// TwinCAT 3 PLC project TcoPneumaticsTests
// Title: TcoPneumaticsTests
// Company: Vortex.Library
// ProjectVersion: 0.6.0.913
// ProgramVersion: 3.1.4024.12
// libraries:
//   Tc2_Standard, * (Beckhoff Automation GmbH)
//   Tc2_System, * (Beckhoff Automation GmbH)
//   Tc3_Module, * (Beckhoff Automation GmbH)
//   TcoCore, 0.6.0.913 (Vortex.Library)
//   TcoPneumatics, 0.6.0.913 (Vortex.Library)
// project tree:
//   ComponentExampleImplementation/ExampleCyclinderUsage/ ExampleCylinderContext.TcPOU
//   ComponentExampleImplementation/ExampleCylinder/ ExampleCylinder.TcPOU, ExampleCylinderConfig.TcDUT, ExampleCylinderMoveTask.TcPOU, ExampleCylinderStatus.TcDUT
//   ComponentExampleImplementation/ EXAMPLE_MAIN.TcPOU
//   GVLs/ IO.TcGVL
//   / PlcTask.TcTTO
//   POUs/CylinderBaseTests/ CylinderBaseImplemented.TcPOU, DoubleCylinderBaseImplemented.TcPOU, CylinderBaseTestContext.TcPOU, DoubleCylinderBaseTestContext.TcPOU, eCyclinderBaseTests.TcDUT
//   POUs/CylinderTests/ DoubleCylinderTestContext.TcPOU, eCyclinderTests.TcDUT, CylinderTestContext.TcPOU
//   POUs/ DefaultContext.TcPOU, MAIN.TcPOU
// (motion and I/O tree: see PLC project tcopneumatics)
// real-time tasks:
//   TASK PlcTask: cycle T#10ms, priority 20, ADS port 350
//   TASK PlcTask1: cycle T#10ms, priority 21, ADS port 351

CONFIGURATION TcoPneumaticsTests
    RESOURCE PLC ON TwinCAT3
        TASK PlcTask(INTERVAL := T#10ms, PRIORITY := 20);
        PROGRAM MAIN WITH PlcTask : MAIN;
        PROGRAM EXAMPLE_MAIN WITH PlcTask : EXAMPLE_MAIN;
    END_RESOURCE
END_CONFIGURATION

// ---- ComponentExampleImplementation/ExampleCylinder/ExampleCylinderConfig.TcDUT
TYPE ExampleCylinderConfig :
STRUCT
    TimeToReachHomePosition : TIME := T#10S;
    TimeToReachWorkPosition : TIME := T#10S;
END_STRUCT
END_TYPE

// ---- ComponentExampleImplementation/ExampleCylinder/ExampleCylinderStatus.TcDUT
TYPE ExampleCylinderStatus :
STRUCT
    ActionDescription : STRING(100);
END_STRUCT
END_TYPE

// ---- POUs/CylinderBaseTests/eCyclinderBaseTests.TcDUT
{attribute 'qualified_only'}
{attribute 'strict'}
TYPE eCyclinderBaseTests :
(
    Invalid := 50,
    GetAtHome := 100,
    GetAtWork := 200
);
END_TYPE

// ---- POUs/CylinderTests/eCyclinderTests.TcDUT
{attribute 'qualified_only'}
{attribute 'strict'}
TYPE eCyclinderTests :
(
    Invalid := 25,
    StopMovement := 50,
    MoveHomeMoving := 100,
    MoveHomeMovingReached := 200,
    MoveWorkMoving := 300,
    MoveWorkMovingReached := 400,
    AbortMoveTask := 500,
    DisableHome := 600,
    DisableWork := 700,
    SuspendHome := 610,
    SuspendWork := 710,
    SuspendHomeInverted := 620,
    SuspendWorkInverted := 720,
    SuspendHomeExpression := 630,
    SuspendWorkExpression := 730
);
END_TYPE

// ---- GVLs/IO.TcGVL
{attribute 'qualified_only'}
VAR_GLOBAL
    {attribute addProperty Name "A1"}
    A1 AT %I* : ARRAY[0..7] OF BOOL;
    {attribute addProperty Name "A2"}
    A2 AT %Q* : ARRAY[0..7] OF BOOL;
END_VAR

// ---- POUs/MAIN.TcPOU
PROGRAM MAIN
VAR
    _defaultContext : DefaultContext;
    _cylinderBaseTests : CylinderBaseTestContext;
    _doubleCylinderBaseTests : DoubleCylinderBaseTestContext;
    _cylinderTests : CylinderTestContext;
    _doubleCylinderTests : DoubleCylinderTestContext;
END_VAR

_defaultContext.Run();
_cylinderTests.ProbeRun();
_doubleCylinderTests.ProbeRun();
_cylinderBaseTests.ProbeRun();
_doublecylinderBaseTests.ProbeRun();

END_PROGRAM

// ---- POUs/DefaultContext.TcPOU
FUNCTION_BLOCK DefaultContext EXTENDS TcoCore.TcoContext
VAR
    {attribute addProperty _moveHomeDefaultName "<#MOVE HOME#>"}
    {attribute addProperty _moveWorkDefaultName "<#MOVE TO WORK#>"}
    {attribute addProperty _stopDefaultName "<#STOP a#>"}
    _wpfCyclinder : TcoPneumatics.TcoCylinder(THIS^);
    {attribute addProperty _moveHomeDefaultName "<#MOVE HOME#>"}
    {attribute addProperty _moveWorkDefaultName "<#MOVE TO WORK#>"}
    {attribute addProperty _stopDefaultName "<#STOPDOUBLE#>"}
    _wpfDoubleCyclinder : TcoPneumatics.TcoDoubleCylinder(THIS^);
    {attribute addProperty NameMoveHomeTask "<#In task#>"}
    _wpfCyclinder_1 : TcoPneumatics.TcoCylinder(THIS^);
    {attribute addProperty NameMoveHomeTask "<#In task#>"}
    _wpfCyclinder_2 : TcoPneumatics.TcoCylinder(THIS^);
    {attribute addProperty NameMoveHomeTask "<#In task#>"}
    _wpfCyclinder_3 : TcoPneumatics.TcoCylinder(THIS^);
    disableSignalWork : BOOL;
    disableSignalHome : BOOL;
    suspendSignalWork : BOOL;
    suspendSignalHome : BOOL;
    refilCondition : BOOL;
END_VAR

METHOD PROTECTED Main
VAR
    ;
END_VAR
THIS^.RtcSynchronize(TRUE, '', 60);
_wpfCyclinder.Service();

_wpfCyclinder(inoAtHomePos := IO.A1[0],
    inoAtWorkPos := IO.A1[1],
    inoToHomePos := IO.A2[0],
    inoToWorkPos := IO.A2[1]);

_wpfCyclinder.AbortMoveHome(disableSignalHome);
_wpfCyclinder.AbortMoveWork(disableSignalWork);
_wpfCyclinder.SuspendMoveHome(suspendSignalHome);
_wpfCyclinder.SuspendMoveWork(suspendSignalWork);
//optional blocking options
//_wpfCyclinder.SuspendMoveWorkInverted(suspendSignalWork);	// is basicaly option how to reproduce exaxt symbol and Not condition
//_wpfCyclinder.SuspendMoveWorkExpression(NOT suspendSignalWork,'Your own msg');	// is basicaly option how to reproduce exaxt symbol and Not condition
_wpfCyclinder.Refill(T#200MS);
_wpfDoubleCyclinder.Service();

_wpfDoubleCyclinder(inoAtHomePos1 := IO.A1[0],
    inoAtHomePos2 := IO.A1[1],
    inoAtWorkPos1 := IO.A1[2],
    inoAtWorkPos2 := IO.A1[3],
    inoToHomePos := IO.A2[3],
    inoToWorkPos := IO.A2[4]);

_wpfDoubleCyclinder.AbortMoveHome(disableSignalHome);
_wpfDoubleCyclinder.AbortMoveWork(disableSignalWork);
_wpfDoubleCyclinder.SuspendMoveHome(suspendSignalHome);
_wpfDoubleCyclinder.SuspendMoveWork(suspendSignalWork);
//optional blocking options
//_wpfDoubleCyclinder.SuspendMoveWorkInverted(suspendSignalWork);	// is basicaly option how to reproduce exaxt symbol and Not condition
//_wpfDoubleCyclinder.SuspendMoveWorkExpression(NOT suspendSignalWork,'Your own msg');	// is basicaly option how to reproduce exaxt symbol and Not condition
_wpfDoubleCyclinder.Refill(T#200MS);
END_METHOD

END_FUNCTION_BLOCK

// ---- POUs/CylinderBaseTests/CylinderBaseTestContext.TcPOU
FUNCTION_BLOCK CylinderBaseTestContext EXTENDS TcoCore._internals_TcoContext
VAR
    _sut : CylinderBaseImplemented(THIS^);
    _sutInvalid : CylinderBaseImplemented(THIS^);
    _atHomeSignal : BOOL;
    _atWorkSignal : BOOL;
    _toHomeSignal : BOOL;
    _toWorkSignal : BOOL;
END_VAR
VAR
    _get_AtHome : BOOL;
    _get_AtWork : BOOL;
END_VAR

METHOD PROTECTED Main
_sut(inoAtHomePos := _atHomeSignal,
    inoAtWorkPos := _atWorkSignal,
    inoToHomePos := _toHomeSignal,
    inoToWorkPos := _toWorkSignal);

CASE _testId OF
    eCyclinderBaseTests.Invalid:
        _sutInvalid.AtHome;
        _sutInvalid.AtWork;
        _sutInvalid.Restore();
        _sutInvalid.Stop();
    eCyclinderBaseTests.GetAtHome:
        _get_AtHome := _sut.AtHome;
    eCyclinderBaseTests.GetAtWork:
        _get_AtWork := _sut.AtWork;
END_CASE
END_METHOD

END_FUNCTION_BLOCK

// ---- POUs/CylinderBaseTests/CylinderBaseImplemented.TcPOU
FUNCTION_BLOCK CylinderBaseImplemented EXTENDS TcoPneumatics.TcoCylinder

SUPER^(inoAtHomePos := inoAtHomePos,
    inoAtWorkPos := inoAtWorkPos,
    inoToHomePos := inoToHomePos,
    inoToWorkPos := inoToWorkPos);

PROPERTY MoveHomeTask : TcoCore.ITcoTask
GET
END_GET
SET
END_SET
END_PROPERTY

PROPERTY MoveWorkTask : TcoCore.ITcoTask
GET
END_GET
SET
END_SET
END_PROPERTY

PROPERTY StopTask : TcoCore.ITcoTask
GET
END_GET
SET
END_SET
END_PROPERTY

END_FUNCTION_BLOCK

// ---- POUs/CylinderBaseTests/DoubleCylinderBaseTestContext.TcPOU
FUNCTION_BLOCK DoubleCylinderBaseTestContext EXTENDS TcoCore._internals_TcoContext
VAR
    _sut : DoubleCylinderBaseImplemented(THIS^);
    _sutInvalid : DoubleCylinderBaseImplemented(THIS^);
    _atHomeSignal : BOOL;
    _atWorkSignal : BOOL;
    _toHomeSignal : BOOL;
    _toWorkSignal : BOOL;
END_VAR
VAR
    _get_AtHome : BOOL;
    _get_AtWork : BOOL;
END_VAR

METHOD PROTECTED Main
_sut(inoAtHomePos1 := _atHomeSignal,
    inoAtHomePos2 := _atHomeSignal,
    inoAtWorkPos1 := _atWorkSignal,
    inoAtWorkPos2 := _atWorkSignal,
    inoToHomePos := _toHomeSignal,
    inoToWorkPos := _toWorkSignal);

CASE _testId OF
    eCyclinderBaseTests.Invalid:
        _sutInvalid.AtHome;
        _sutInvalid.AtWork;
        _sutInvalid.Restore();
        _sutInvalid.Stop();
    eCyclinderBaseTests.GetAtHome:
        _get_AtHome := _sut.AtHome;
    eCyclinderBaseTests.GetAtWork:
        _get_AtWork := _sut.AtWork;
END_CASE
END_METHOD

END_FUNCTION_BLOCK

// ---- POUs/CylinderBaseTests/DoubleCylinderBaseImplemented.TcPOU
FUNCTION_BLOCK DoubleCylinderBaseImplemented EXTENDS TcoPneumatics.TcoDoubleCylinderBase

SUPER^(inoAtHomePos1 := inoAtHomePos1,
    inoAtHomePos2 := inoAtHomePos2,
    inoAtWorkPos1 := inoAtWorkPos1,
    inoAtWorkPos2 := inoAtWorkPos2,
    inoToHomePos := inoToHomePos,
    inoToWorkPos := inoToWorkPos);

PROPERTY MoveHomeTask : TcoCore.ITcoTask
GET
END_GET
SET
END_SET
END_PROPERTY

PROPERTY MoveWorkTask : TcoCore.ITcoTask
GET
END_GET
SET
END_SET
END_PROPERTY

PROPERTY StopTask : TcoCore.ITcoTask
GET
END_GET
SET
END_SET
END_PROPERTY

END_FUNCTION_BLOCK

// ---- POUs/CylinderTests/CylinderTestContext.TcPOU
FUNCTION_BLOCK CylinderTestContext EXTENDS TcoCore._internals_TcoContext
VAR
    {attribute addProperty _moveHomeDefaultName "<#MOVE HOME SWEET HOME#>"}
    {attribute addProperty _moveWorkDefaultName "<#MOVE TO WORK HARD WORK#>"}
    {attribute addProperty _stopDefaultName "<#STOP AND THINK#>"}
    _sut : TcoPneumatics.TcoCylinder(THIS^);
    _sutInvalid : TcoPneumatics.TcoCylinder(THIS^);
    _atHomeSignal : BOOL;
    _moveHomeSignal : BOOL;
    _atWorkSignal : BOOL;
    _moveWorkSignal : BOOL;
END_VAR
VAR
    _moveHomeDone : BOOL;
    _moveWorkDone : BOOL;
    _disableSignal : BOOL;
    _suspendSignal : BOOL;
    _expresionMessage : STRING;
END_VAR

METHOD PROTECTED Main
_sut(inoAtHomePos := _atHomeSignal,
    inoAtWorkPos := _atWorkSignal,
    inoToHomePos := _moveHomeSignal,
    inoToWorkPos := _moveWorkSignal);

CASE _testId OF
    eCyclinderTests.Invalid:
        _sutInvalid.Stop();
        _sutInvalid.MoveToHome();
        _sutInvalid.MoveToWork();
        _sutInvalid.Service();
        _sutInvalid.AtHome;
        _sutInvalid.AtWork;
        _sutInvalid.AbortMoveHome(_disableSignal);
        _sutInvalid.AbortMoveHome(_disableSignal);
        _sutInvalid.Config.TimeToReachHomePosition := T#1MS;
        _sutInvalid.Config.TimeToReachWorkPosition := T#1MS;
        _sutInvalid.Status.ActionDescription;
    eCyclinderTests.StopMovement:
        _sut.Stop();
    eCyclinderTests.MoveHomeMoving:
        _moveHomeDone := _sut.MoveToHome().Done;
    eCyclinderTests.MoveHomeMovingReached:
        _moveHomeDone := _sut.MoveToHome().Done;
    eCyclinderTests.MoveWorkMoving:
        _moveWorkDone := _sut.MoveToWork().Done;
    eCyclinderTests.MoveWorkMovingReached:
        _moveWorkDone := _sut.MoveToWork().Done;
    eCyclinderTests.AbortMoveTask:
        _sut.MoveHomeTask.Abort();
    eCyclinderTests.DisableHome:
        _sut.AbortMoveHome(_disableSignal);
    eCyclinderTests.DisableWork:
        _sut.AbortMoveWork(_disableSignal);
    eCyclinderTests.SuspendHome:
        _sut.SuspendMoveHome(_suspendSignal);
    eCyclinderTests.SuspendWork:
        _sut.SuspendMoveWork(_suspendSignal);
    eCyclinderTests.SuspendHomeInverted:
        _sut.SuspendMoveHomeInverted(_suspendSignal);
    eCyclinderTests.SuspendWorkInverted:
        _sut.SuspendMoveWorkInverted(_suspendSignal);
    eCyclinderTests.SuspendHomeExpression:
        _sut.SuspendMoveHomeExpression(_suspendSignal, _expresionMessage);
    eCyclinderTests.SuspendWorkExpression:
        _sut.SuspendMoveWorkExpression(_suspendSignal, _expresionMessage);
END_CASE
END_METHOD

END_FUNCTION_BLOCK

// ---- POUs/CylinderTests/DoubleCylinderTestContext.TcPOU
FUNCTION_BLOCK DoubleCylinderTestContext EXTENDS TcoCore._internals_TcoContext
VAR
    {attribute addProperty _moveHomeDefaultName "<#MOVE HOME SWEET HOME#>"}
    {attribute addProperty _moveWorkDefaultName "<#MOVE TO WORK HARD WORK#>"}
    {attribute addProperty _stopDefaultName "<#STOP AND THINK#>"}
    _sut : TcoPneumatics.TcoDoubleCylinder(THIS^);
    _sutInvalid : TcoPneumatics.TcoDoubleCylinder(THIS^);
    _atHomeSignal : BOOL;
    _moveHomeSignal : BOOL;
    _atWorkSignal : BOOL;
    _moveWorkSignal : BOOL;
END_VAR
VAR
    _moveHomeDone : BOOL;
    _moveWorkDone : BOOL;
    _disableSignal : BOOL;
    _suspendSignal : BOOL;
    _expresionMessage : STRING;
END_VAR

METHOD PROTECTED Main
_sut(inoAtHomePos1 := _atHomeSignal,
    inoAtHomePos2 := _atHomeSignal,
    inoAtWorkPos1 := _atWorkSignal,
    inoAtWorkPos2 := _atWorkSignal,
    inoToHomePos := _moveHomeSignal,
    inoToWorkPos := _moveWorkSignal);

CASE _testId OF
    eCyclinderTests.Invalid:
        _sutInvalid.Stop();
        _sutInvalid.MoveToHome();
        _sutInvalid.MoveToWork();
        _sutInvalid.Service();
        _sutInvalid.AtHome;
        _sutInvalid.AtWork;
        _sutInvalid.AbortMoveHome(_disableSignal);
        _sutInvalid.AbortMoveHome(_disableSignal);
        _sutInvalid.Config.TimeToReachHomePosition := T#1MS;
        _sutInvalid.Config.TimeToReachWorkPosition := T#1MS;
        _sutInvalid.Status.ActionDescription;
    eCyclinderTests.StopMovement:
        _sut.Stop();
    eCyclinderTests.MoveHomeMoving:
        _moveHomeDone := _sut.MoveToHome().Done;
    eCyclinderTests.MoveHomeMovingReached:
        _moveHomeDone := _sut.MoveToHome().Done;
    eCyclinderTests.MoveWorkMoving:
        _moveWorkDone := _sut.MoveToWork().Done;
    eCyclinderTests.MoveWorkMovingReached:
        _moveWorkDone := _sut.MoveToWork().Done;
    eCyclinderTests.AbortMoveTask:
        _sut.MoveHomeTask.Abort();
    eCyclinderTests.DisableHome:
        _sut.AbortMoveHome(_disableSignal);
    eCyclinderTests.DisableWork:
        _sut.AbortMoveWork(_disableSignal);
    eCyclinderTests.SuspendHome:
        _sut.SuspendMoveHome(_suspendSignal);
    eCyclinderTests.SuspendWork:
        _sut.SuspendMoveWork(_suspendSignal);
    eCyclinderTests.SuspendHomeInverted:
        _sut.SuspendMoveHomeInverted(_suspendSignal);
    eCyclinderTests.SuspendWorkInverted:
        _sut.SuspendMoveWorkInverted(_suspendSignal);
    eCyclinderTests.SuspendHomeExpression:
        _sut.SuspendMoveHomeExpression(_suspendSignal, _expresionMessage);
    eCyclinderTests.SuspendWorkExpression:
        _sut.SuspendMoveWorkExpression(_suspendSignal, _expresionMessage);
END_CASE
END_METHOD

END_FUNCTION_BLOCK

// ---- ComponentExampleImplementation/EXAMPLE_MAIN.TcPOU
PROGRAM EXAMPLE_MAIN
VAR
    _context : ExampleCylinderContext;
END_VAR

_context.Run();

END_PROGRAM

// ---- ComponentExampleImplementation/ExampleCyclinderUsage/ExampleCylinderContext.TcPOU
FUNCTION_BLOCK ExampleCylinderContext EXTENDS TcoCore.TcoContext
VAR
    _exampleCylinder : ExampleCylinder(THIS^);
    _atHome : BOOL;
    _atWork : BOOL;
    _toHome : BOOL;
    _toWork : BOOL;
END_VAR

(*~
    <docu>
        <summary>
            Main method of the TcoContext. This is the entry point of any control logic that belongs to this context.
            The call of this method is ensured by calling the <c>InstanceName.Run()</c> method, and it must not be called explicitly.
            This method is abstract, and it must be overridden in derived block.
        </summary>
    </docu>
~*)
METHOD PROTECTED Main
VAR_INST
    _state : INT;
END_VAR
_exampleCylinder(inoAtHomePos := _atHome,
    inoAtWorkPos := _atWork,
    inoToHomePos := _toHome,
    inoToWorkPos := _toWork);

CASE _state OF
    0:
        IF (_exampleCylinder.MoveToHome().Done) THEN
            _state := 10;
        END_IF
    10:
        IF (_exampleCylinder.MoveToWork().Done) THEN
            _state := 0;
        END_IF
END_CASE
END_METHOD

END_FUNCTION_BLOCK

// ---- ComponentExampleImplementation/ExampleCylinder/ExampleCylinder.TcPOU
(*~
        <docu>
            <summary>
                This is an example implementation of `ExampleCyclinder` component.
            </summary>
        </docu>
~*)
FUNCTION_BLOCK ExampleCylinder EXTENDS TcoCore.TcoComponent
VAR_IN_OUT
    (*~
        <docu>
            <summary>
                Home position sensor.
            </summary>
        </docu>
    ~*)
    {attribute addProperty Name "<#Home position sensor#>"}
    inoAtHomePos : BOOL;
    (*~
        <docu>
            <summary>
                Working position sensor.
            </summary>
        </docu>
    ~*)
    {attribute addProperty Name "<#Work position sensor#>"}
    inoAtWorkPos : BOOL;
    (*~
        <docu>
            <summary>
                Move to working home position signal.
            </summary>
        </docu>
    ~*)
    {attribute addProperty Name "<#Move to home position actuator#>"}
    inoToHomePos : BOOL;
    (*~
        <docu>
            <summary>
                Move to working posistion signal.
            </summary>
        </docu>
    ~*)
    {attribute addProperty Name "<#Move to work position actuator#>"}
    inoToWorkPos : BOOL;
END_VAR
VAR
    (*~
        <docu>
            <summary>
                Home position sensor.
            </summary>
        </docu>
    ~*)
    {attribute addProperty Name "<#Home position sensor#>"}
    _atHomePos : BOOL;
    (*~
        <docu>
            <summary>
                Working position sensor.
            </summary>
        </docu>
    ~*)
    {attribute addProperty Name "<#Work position sensor#>"}
    _atWorkPos : BOOL;
    (*~
        <docu>
            <summary>
                Move to working home position signal.
            </summary>
        </docu>
    ~*)
    {attribute addProperty Name "<#Move to home position actuator#>"}
    _toHomePos : BOOL;
    (*~
        <docu>
            <summary>
                Move to working posistion signal.
            </summary>
        </docu>
    ~*)
    {attribute addProperty Name "<#Move to work position actuator#>"}
    _toWorkPos : BOOL;
END_VAR
VAR
    _atHomePosSignalInfo : TcoCore.TcoSignalInfo;
    _atWorkPosSignalInfo : TcoCore.TcoSignalInfo;
    _toHomePosSignalInfo : TcoCore.TcoSignalInfo;
    _toWorkPosSignalInfo : TcoCore.TcoSignalInfo;
END_VAR
VAR
    {attribute addProperty Name "<#Move Home#>"}
    _moveHomeDefault : ExampleCylinderMoveTask(THIS^);
    {attribute addProperty Name "<#Move to Work#>"}
    _moveWorkDefault : ExampleCylinderMoveTask(THIS^);
    {attribute addProperty Name "<#Stop#>"}
    _stopDefault : TcoCore.TcoTask(THIS^);
END_VAR
VAR
    _config : TcoCylinderConfig;
    _status : TcoCylinderStatus;
END_VAR

// Updates I/O
UpdateIO();
// Disables mutualy exclusive actions
_moveWorkDefault.Enabled := NOT _moveHomeDefault.Busy;

_moveHomeDefault(PositionSensor := _atHomePos,
    MoveToPositionSignal := _toHomePos,
    InverseSignal := _toWorkPos,
    MaxTimeToReachPosition := _config.TimeToReachHomePosition,
    PositionName := '<#Home#>');
// Disables mutualy exclusive actions
_moveHomeDefault.Enabled := NOT _moveWorkDefault.Busy;

_moveWorkDefault(PositionSensor := _atWorkPos,
    MoveToPositionSignal := _toWorkPos,
    InverseSignal := _toHomePos,
    MaxTimeToReachPosition := _config.TimeToReachWorkPosition,
    PositionName := '<#Work#>');

IF (_stopDefault.Execute()) THEN
    _toHomePos := FALSE;
    _toWorkPos := FALSE;
    _moveHomeDefault.Abort();
    _moveWorkDefault.Abort();
    _stopDefault.Abort();
    _moveHomeDefault.Restore();
    _moveWorkDefault.Restore();
    _stopDefault.Restore();
    _stopDefault.DoneWhen(TRUE);
END_IF

// For further discussion about Status
IF (_moveHomeDefault.Busy) THEN
    _status.ActionDescription := 'Moving to home position';
ELSIF (_moveWorkDefault.Busy) THEN
    _status.ActionDescription := 'Moving to work position';
ELSIF (_stopDefault.Busy) THEN
    _status.ActionDescription := 'Stopping pressure';
ELSE
    _status.ActionDescription := 'Idle';
END_IF

UpdateIO();

(*~
    <docu>
        <summary>
            Gets whether the piston is in home position.
        </summary>
    </docu>
~*)
PROPERTY AtHome : bool
GET
AtHome := THIS^._atHomePos;
END_GET
END_PROPERTY

(*~
    <docu>
        <summary>
            Gets whether the piston is in work position.
        </summary>
    </docu>
~*)
PROPERTY AtWork : bool
GET
AtWork := _atWorkPos;
END_GET
END_PROPERTY

(*~
    <docu>
        <summary>
            Gets the configuration of the cylinder.
        </summary>
    </docu>
~*)
PROPERTY Config : REFERENCE TO TcoCylinderConfig
GET
Config REF= config;
END_GET
END_PROPERTY

(*~
    <docu>
        <summary>
            Gets the `MoveHomeTask` task that controls the moving of the cyclinder in home position.
        </summary>
    </docu>
~*)
PROPERTY MoveHomeTask : TcoCore.ITcoTask
GET
MoveHomeTask := _moveHomeDefault;
END_GET
END_PROPERTY

(*~
    <docu>
        <summary>
            Starts movement into home position.
        </summary>
    </docu>
~*)
METHOD MoveToHome : TcoCore.ITcoTaskStatus
IF (MoveHomeTask <> 0) THEN
    MoveToHome := MoveHomeTask.Invoke();
END_IF;
END_METHOD

(*~
    <docu>
        <summary>
            Starts movement into work position.
        </summary>
    </docu>
~*)
METHOD MoveToWork : TcoCore.ITcoTaskStatus
IF (MoveWorkTask <> 0) THEN
    MoveToWork := MoveWorkTask.Invoke();
END_IF;
END_METHOD

(*~
    <docu>
        <summary>
            Gets the `MoveWorkTask` task that controls the moving of the cyclinder into work position.
        </summary>
    </docu>
~*)
PROPERTY MoveWorkTask : TcoCore.ITcoTask
GET
MoveWorkTask := _moveWorkDefault;
END_GET
END_PROPERTY

(*~
    <docu>
        <summary>
            Restores this instance to the Ready state. Can be called explicitly or from within one of the restore mechanisms.
        </summary>
    </docu>
~*)
METHOD Restore : ITcoRestorable
IF (MoveHomeTask <> 0) THEN
    MoveHomeTask.Restore();
END_IF;

IF (MoveWorkTask <> 0) THEN
    MoveWorkTask.Restore();
END_IF;

IF (StopTask <> 0) THEN
    StopTask.Restore();
END_IF;
END_METHOD

(*~
    <docu>
        <summary>
            Custom service (manual, maintenance) logic.
            This method must be implemented in derived class.
        </summary>
    </docu>
~*)
METHOD PROTECTED ServiceMode
END_METHOD

PROPERTY Status : REFERENCE TO TcoCylinderStatus
GET
Status REF= _status;
END_GET
END_PROPERTY

(*~
    <docu>
        <summary>
            Stops cyclinder movement.
             <remarks>
                <note type="important">
                    This method switched off the signals for the movement of the piston in both direction.
                    However depending on the pnemumatics configuration the movement may contintue if designed in that way.
                    THIS IS NOT A SAFETY FUCTION!
                </note>
            </remarks>
        </summary>
    </docu>
~*)
METHOD Stop : TcoCore.ITcoTaskStatus
IF (StopTask <> 0) THEN
    Stop := StopTask.Invoke();
END_IF;
END_METHOD

(*~
    <docu>
        <summary>
            Gets the `StopTask` task that controls the stopping of the cyclinder.
        </summary>
    </docu>
~*)
PROPERTY StopTask : TcoCore.ITcoTask
GET
StopTask := _stopDefault;
END_GET
END_PROPERTY

METHOD PRIVATE UpdateIO
IF (__ISVALIDREF(inoAtHomePos)) THEN
    _atHomePos := inoAtHomePos;
    _atHomePosSignalInfo.GetSignalInfo(SIZEOF(inoAtHomePos), ADR(inoAtHomePos));
END_IF;

IF (__ISVALIDREF(inoAtWorkPos)) THEN
    _atWorkPos := inoAtWorkPos;
    _atWorkPosSignalInfo.GetSignalInfo(SIZEOF(inoAtWorkPos), ADR(inoAtWorkPos));
END_IF;

IF (__ISVALIDREF(inoToHomePos)) THEN
    inoToHomePos := _toHomePos;
    _toHomePosSignalInfo.GetSignalInfo(SIZEOF(inoToHomePos), ADR(inoToHomePos));
END_IF;

IF (__ISVALIDREF(inoToWorkPos)) THEN
    inoToWorkPos := _toWorkPos;
    _toWorkPosSignalInfo.GetSignalInfo(SIZEOF(inoToWorkPos), ADR(inoToWorkPos));
END_IF;
END_METHOD

END_FUNCTION_BLOCK

// ---- ComponentExampleImplementation/ExampleCylinder/ExampleCylinderMoveTask.TcPOU
FUNCTION_BLOCK ExampleCylinderMoveTask EXTENDS TcoCore.TcoTask
VAR_INPUT
    PositionSensor : BOOL;
    MaxTimeToReachPosition : TIME := T#10S;
    PositionName : STRING(25);
END_VAR
VAR_IN_OUT
    MoveToPositionSignal : BOOL;
    InverseSignal : BOOL;
END_VAR
VAR
    _stringBuilder : TcoCore.StringBuilder;
END_VAR

IF (THIS^.Execute()) THEN
    IF (THIS^.ElapsedTime > MaxTimeToReachPosition) THEN
        THIS^.Messenger.Warning(_stringBuilder.Clear().Append(PositionName).Append(' sensor not reached yet.').ToString());
    END_IF;

    InverseSignal := FALSE;
    MoveToPositionSignal := TRUE;
    THIS^.DoneWhen(PositionSensor);
END_IF

METHOD PUBLIC FB_init : BOOL
VAR_INPUT
    bInitRetains : BOOL; // if TRUE, the retain variables are initialized (warm start / cold start)
    bInCopyCode : BOOL; // if TRUE, the instance afterwards gets moved into the copy code (online change)
    ParentObject : ITcoObject;
END_VAR
END_METHOD

(*~
    <docu>
        <summary>
            Executes when task is aborted.
        </summary>
    </docu>
~*)
METHOD PROTECTED OnAbort
MoveToPositionSignal := FALSE;
END_METHOD

METHOD PROTECTED OnError
END_METHOD

END_FUNCTION_BLOCK
